// TIA Portal project "py_opc" (V16)

(* hardware
DEVICE "PC-System_1"  SIMATIC PC station
   slot 0: "SIMATIC PC station"  Rail  SIMATIC PC-Station  V1.0
      slot 125: "Stationmanager"  Station_Manager  V6.0.4
   slot 1: "HMI_RT_1"  WinCC RT Advanced  6AV2 104-0xxxx-xxxx  16.0.0.0
      slot 33792: "Computer interface"  Host interface
   slot 2: "IE general_1"  IE General  IE_CP  V8.2.0
*)

(* ===== HMI "HMI_RT_1" =====
system functions are stored by id; their names below are inferred from use
connection "Connection_1": OPC, OPC_UA

HMI tags "Default tag table"
   "p1_sel" : Boolean AT ns=gesture_control;i=2, 500 ms
   "p2_sel" : Boolean AT ns=gesture_control;i=3, 500 ms
   "p3_sel" : Boolean AT ns=gesture_control;i=4, 500 ms
   "p1_cmd" : Boolean AT ns=gesture_control;i=5, 500 ms
   "p2_cmd" : Boolean AT ns=gesture_control;i=6, 500 ms
   "p3_cmd" : Boolean AT ns=gesture_control;i=7, 500 ms
   "rotate" : Int, internal

graphic list "pump_rot": 0 'Graphic_10'; 1 'Graphic_11'; 2 'Graphic_12'; 3 'Graphic_13'

screen "Screen_1" 1366x768
   on GenerateScreen: function_f9c01323("rotate", 1, 3, 0, 1)
   GraphicView "Graphic view_6" at 65,208 size 134x134; Picture "Graphic_19"
   GraphicIOField "Graphic I/O field_1" at 70,212 size 124x126; PictureList "pump_rot"
      ProcessValue <- "rotate"
   GraphicView "Graphic view_1" at 65,208 size 134x134; Picture "Graphic_14"
      Visibility <- "p1_cmd"
   GraphicView "Graphic view_2" at 284,208 size 134x134; Picture "Graphic_19"
   GraphicIOField "Graphic I/O field_2" at 289,212 size 124x126; PictureList "pump_rot"
      ProcessValue <- "rotate"
   GraphicView "Graphic view_3" at 284,208 size 134x134; Picture "Graphic_14"
      Visibility <- "p2_cmd"
   GraphicView "Graphic view_4" at 504,208 size 134x134; Picture "Graphic_19"
   GraphicIOField "Graphic I/O field_3" at 509,212 size 124x126; PictureList "pump_rot"
      ProcessValue <- "rotate"
   GraphicView "Graphic view_5" at 504,208 size 134x134; Picture "Graphic_14"
      Visibility <- "p3_cmd"
   IOField "I/O field_1" at 1066,733 size 22x25; FormatPattern 1
      ProcessValue <- "p1_sel"
   IOField "I/O field_2" at 1091,733 size 22x25; FormatPattern 1
      ProcessValue <- "p1_cmd"
   IOField "I/O field_3" at 1146,733 size 22x25; FormatPattern 1
      ProcessValue <- "p2_sel"
   IOField "I/O field_4" at 1172,733 size 22x25; FormatPattern 1
      ProcessValue <- "p2_cmd"
   IOField "I/O field_5" at 1222,733 size 22x25; FormatPattern 1
      ProcessValue <- "p3_sel"
   IOField "I/O field_6" at 1248,733 size 22x25; FormatPattern 1
      ProcessValue <- "p3_cmd"
   TextField "Text field_1" at 43,7 size 402x59; Text 'Gesture Control'
   TextField "Text field_3" at 43,67 size 626x27; Text 'a hobby project on WinCC RT Advanced & Python - by Kamal Lal'
   Button "Button_1" at 1290,722 size 54x39; TextOff 'Q'
      on Click: StopRuntime(0)
   Group "Group" at 65,208 size 134x134; Picture "Graphic_19"; PictureList "pump_rot"
   Group "Group_1" at 284,208 size 134x134; Picture "Graphic_19"; PictureList "pump_rot"
   Group "Group_2" at 504,208 size 134x134; Picture "Graphic_19"; PictureList "pump_rot"
   TextField "Text field_2" at 65,164 size 134x35; Text 'FAN - 1'
      Appearance <- "p1_sel"
   TextField "Text field_4" at 284,164 size 134x35; Text 'FAN - 2'
      Appearance <- "p2_sel"
   TextField "Text field_5" at 504,164 size 134x35; Text 'FAN - 3'
      Appearance <- "p3_sel"
   Group "Group_3" at 791,137 size 368x127
   Group "Group_4" at 41,406 size 621x230
   Button "Button_2" at 985,719 size 54x39; TextOff 'R'
      on Click: ResetBit("p1_cmd"); ResetBit("p2_cmd"); ResetBit("p3_cmd"); ResetBit("p1_sel"); ResetBit("p2_sel"); ResetBit("p3_sel")
   TextField "Text field_9" at 51,595 size 241x22; Text 'OS - Windows 7 Ult. (64 bit)'
   TextField "Text field_14" at 51,491 size 227x22; Text 'Neural Network trained on:'
   TextField "Text field_10" at 341,447 size 275x22; Text 'Communicaion channel - OPC UA'
   TextField "Text field_13" at 341,422 size 226x22; Text 'ML integration with WinCC:'
   TextField "Text field_12" at 341,491 size 239x22; Text 'Machine Learning (ML) logic:'
   TextField "Text field_7" at 51,447 size 271x22; Text 'SIEMENS WinCC Advanced - V16'
   TextField "Text field_11" at 51,422 size 113x22; Text 'Visualization:'
   TextField "Text field_18" at 51,517 size 205x22; Text 'Processor - Intel Core i7'
   TextField "Text field_19" at 51,543 size 130x22; Text 'Memory - 32GB'
   TextField "Text field_20" at 51,569 size 98x22; Text 'GPU - none'
   TextField "Text field_21" at 341,517 size 191x22; Text 'Language - Python 3.7'
   TextField "Text field_22" at 341,543 size 297x22; Text 'Image processing library - OpenCV'
   TextField "Text field_23" at 341,569 size 312x22; Text 'Machine Learning library - Tensorflow'
   TextField "Text field_6" at 797,145 size 99x22; Text 'Operation:'
   TextField "Text field_15" at 821,172 size 325x22; Text '• Showing 1, 2 or 3 selects the device.'
   TextField "Text field_16" at 821,202 size 322x22; Text '• 'PALM OPENING' gesture turns it On.'
   TextField "Text field_17" at 821,232 size 322x22; Text '• 'PALM CLOSING' gesture turns it Off.'
*)